// Block: PPrgArchive8

DATA_BLOCK PPrgArchive8
VERSION : 0.1
   NON_RETAIN
   VAR
      PRG : Array[701..800] of PPrg_Data;
   END_VAR

BEGIN
   // No initialization required
END_DATA_BLOCK
